(* CoDeSys 2.3 library: TcNciUtilities.lib *)
(* Libraries: TcNci.lib 16.11.12 16:23:10, TcMC.lib 18.1.10 08:53:12, TcBaseMath.lib 27.7.04 11:07:56, TcMath.lib 23.9.04 14:15:30, TcNC.lib 10.10.08 16:55:34, TcIoFunctions.lib 21.7.11 16:19:20, TcUtilities.lib 2.3.12 18:25:40, TcSystem.lib 27.2.12 14:08:36, TcBase.lib 14.5.09 11:14:08, standard.lib 5.6.98 11:03:02, TcNcCfg.lib 22.9.03 17:16:34 *)

(* POU MAIN, ST *)
PROGRAM MAIN
VAR
END_VAR
;
END_PROGRAM

(* POU F_GetVersionTcNciUtilities, ST *)
FUNCTION F_GetVersionTcNciUtilities : UINT
VAR_INPUT
	nVersionElement	: INT;
END_VAR
(*
	Possible nVersionElement parameter:
	1	:	major number
	2	:	minor number
	3	:	revision number
*)
(* Version history:
Date        | Version   | created with							| Author				| Remark
-----------------------------------------------------------------------------------------------------------------------------------------------------------------------------------------------------------------
2013-01-10  | 1.0.3     | TC 2.11								| bw					| Default ADS timeout added
-----------------------------------------------------------------------------------------------------------------------------------------------------------------------------------------------------------------
2013-01-10  | 1.0.2     | TC 2.11 saved as 2.11 Lib		| kbn					| 
-----------------------------------------------------------------------------------------------------------------------------------------------------------------------------------------------------------------
2003-10-07  | 1.0.1     | TC 2.9 B947 saved as 2.8 Lib	| kbn					| lib includes
-----------------------------------------------------------------------------------------------------------------------------------------------------------------------------------------------------------------
2003-09-02  | 1.0.0     | TC 2.9 B947 saved as 2.8 Lib	| Christoph C.		| first release
-----------------------------------------------------------------------------------------------------------------------------------------------------------------------------------------------------------------
*)
CASE nVersionElement OF
1:	(* major number *)
	F_GetVersionTcNciUtilities := 1;
2:	(* minor number *)
	F_GetVersionTcNciUtilities := 0;
3:	(* revision number *)
	F_GetVersionTcNciUtilities := 3;
ELSE
	F_GetVersionTcNciUtilities := 16#FFFF;
END_CASE
END_FUNCTION

(* POU ItpPpgAppendGenericBlock, ST *)
(* Name:       ItpPpgAppendGenericBlock                     *)
(* Desc:       append generic block to the part program     *)
(*             this is just a beta implementation & subject *)
(*             to change                                    *)
(* Author:     kbn                                          *)
(* Date:       05-November-2002                             *)
(* Revision:   VER 1.0.1                                    *)
(* last edit:	VER 1.0.3                                    *)
(*==========================================================*)

FUNCTION_BLOCK ItpPpgAppendGenericBlock
VAR_INPUT
	bExecute:	BOOL;
	sPathName:	STRING;	(* contains path & file name *)
	sBlock:		STRING;
	tTimeOut:	TIME	:= DEFAULT_ADS_TIMEOUT;
END_VAR
VAR_OUTPUT
	bBusy:		BOOL;
	bErr:			BOOL;
	nErrId:		UDINT;
END_VAR
VAR
	nState:				UDINT	:= 0;
	nErrState:			UDINT	:= 0;
	hFile:				UINT;
	fbFileOpen:			FB_FileOpen;
	fbFileClose:		FB_FileClose;
	fbFileAppendLine:	FB_FilePuts;
END_VAR
CASE nState OF
0:
	IF bExecute THEN
		bBusy			:= TRUE;
		bErr			:= FALSE;
		nErrId		:= 0;
		nErrState	:= 0;
		hFile			:= 0;

		(* open existing file *)
		fbFileOpen(
			sNetId		:= '',
			sPathName	:= sPathName,
			nMode			:= FOPEN_MODEAPPEND OR FOPEN_MODETEXT,
			ePath			:= PATH_GENERIC,
			bExecute		:= TRUE,
			tTimeout		:= tTimeOut );

		nState	:= 10;
	END_IF

10:
	(* open existing file *)
	fbFileOpen();

	IF NOT fbFileOpen.bBusy THEN
		fbFileOpen( bExecute := FALSE );
		IF NOT fbFileOpen.bError THEN
			hFile	:= fbFileOpen.hFile;

			(* append line *)
			fbFileAppendLine(
				sNetId	:= '',
				hFile		:= hFile,
				sLine		:= sBlock,
				bExecute	:= TRUE,
				tTimeout	:= tTimeOut );

			nState	:= 20;
		ELSE
			bErr		:= TRUE;
			nErrId	:= fbFileOpen.nErrId;
			nErrState:= nState;
			nState	:= 9999;
		END_IF
	END_IF

20:
	(* append line *)
	fbFileAppendLine();

	IF NOT fbFileAppendLine.bBusy THEN
		fbFileAppendLine( bExecute := FALSE );
		IF NOT fbFileAppendLine.bError THEN
			fbFileClose(
				sNetId	:= '',
				hFile		:= hFile,
				bExecute	:= TRUE,
				tTimeout	:= tTimeOut );
			nState	:= 30;
		ELSE
			bErr		:= TRUE;
			nErrId	:= fbFileAppendLine.nErrId;
			nErrState	:= nState;
			nState	:= 30;	(* we have to close the file anyway *)
		END_IF
	END_IF

30:
	(* close file again *)
	fbFileClose(
		sNetId	:= '',
		hFile		:= hFile,
		bExecute	:= TRUE,
		tTimeout	:= tTimeOut );

	IF NOT fbFileClose.bBusy THEN
		fbFileClose( bExecute := FALSE );
		IF NOT fbFileClose.bError THEN
			IF NOT bExecute THEN
				nState	:= 0;
			ELSE
				nState	:= 9999;
			END_IF
			bBusy	:= FALSE;
		ELSE
			bErr		:= TRUE;
			nErrId	:= fbFileClose.nErrId;
			nErrState:= nState;
			nState	:= 9999;
		END_IF
	END_IF

9999:
	fbFileOpen( bExecute := FALSE );
	fbFileAppendLine( bExecute := FALSE );
	fbFileClose( bExecute := FALSE );

	bBusy	:= FALSE;

	IF NOT bExecute THEN
		nState	:= 0;
	END_IF


END_CASE
END_FUNCTION_BLOCK

(* POU ItpPpgAppendGeoCircleByRadius, ST *)
(* Name:       ItpPpgAppendGeoCircleByRadius                *)
(* Desc:       append a  circle to part program             *)
(*             this is just a beta implementation & subject *)
(*             to change                                    *)
(* Author:     kbn                                          *)
(* Date:       05-November-2002                             *)
(* Revision:   VER 1.0.1                                    *)
(* last edit:	VER 1.0.3                                    *)
(*==========================================================*)

FUNCTION_BLOCK ItpPpgAppendGeoCircleByRadius
VAR_INPUT
	bExecute:		BOOL;
	sPathName:		STRING;	(* contains path & file name *)
	bClockWise:		BOOL;
	fTargetXPos:	LREAL;
	fTargetYPos:	LREAL;
	fTargetZPos:	LREAL;
	fRadius:			LREAL;
	fPathVelo:		LREAL;
	nBlockNo:		UDINT;
	tTimeOut:		TIME	:= DEFAULT_ADS_TIMEOUT;
END_VAR
VAR_OUTPUT
	bBusy:		BOOL;
	bErr:			BOOL;
	nErrId:		UDINT;
END_VAR
VAR
	nState:				UDINT	:= 0;
	fbFormatString:	FB_FormatString;
	sBlock:				T_MaxString;
	fbAppendBlock:		ItpPpgAppendGenericBlock;
	fBlockNo:			LREAL;
END_VAR
CASE nState OF

0:
	IF bExecute THEN
		bBusy		:= TRUE;
		bErr		:= FALSE;
		nErrId	:= 0;

		fBlockNo	:= UDINT_TO_LREAL( nBlockNo );

		IF bClockWise THEN
			fbFormatString(
				sFormat:= 'N%.0f G2 X%.3f Y%.3f Z%.3f B%.3f F%.3f $N',
				arg1:= F_LREAL( fBlockNo ),
				arg2:= F_LREAL( fTargetXPos ),
				arg3:= F_LREAL( fTargetYPos ),
				arg4:= F_LREAL( fTargetZPos ),
				arg5:= F_LREAL( fRadius ),
				arg6:= F_LREAL( fPathVelo ) );
		ELSE
			fbFormatString(
				sFormat:= 'N%.0f G3 X%.3f Y%.3f Z%.3f B%.3f F%.3f $N',
				arg1:= F_LREAL( fBlockNo ),
				arg2:= F_LREAL( fTargetXPos ),
				arg3:= F_LREAL( fTargetYPos ),
				arg4:= F_LREAL( fTargetZPos ),
				arg5:= F_LREAL( fRadius ),
				arg6:= F_LREAL( fPathVelo ) );
		END_IF

		IF NOT fbFormatString.bError THEN
			sBlock	:= fbFormatString.sOut;

			nState	:= 10;
		ELSE
			bErr		:= TRUE;
			nErrId	:= fbFormatString.nErrId;

			nState	:= 9999;
		END_IF

	END_IF

10:
	fbAppendBlock(
		bExecute		:= TRUE,
		sPathName	:= sPathName,
		sBlock		:= sBlock,
		tTimeOut		:= tTimeOut );

	IF NOT fbAppendBlock.bBusy THEN
		fbAppendBlock( bExecute := FALSE );

		IF NOT fbAppendBlock.bErr THEN
			bBusy	:= FALSE;
			IF NOT bExecute THEN
				nState	:= 0;
			ELSE
				nState	:= 9999;
			END_IF
		ELSE
			(* an error occured *)
			bErr		:= TRUE;
			nErrId	:= fbAppendBlock.nErrId;
			nState	:= 9999;
		END_IF

	END_IF

9999:
	bBusy	:= FALSE;
	fbAppendBlock( bExecute := FALSE );

	IF NOT bExecute THEN
		nState	:= 0;
	END_IF

END_CASE
END_FUNCTION_BLOCK

(* POU ItpPpgAppendGeoLine, ST *)
(* Name:       ItpPpgAppendGeoLine                          *)
(* Desc:       append a line to the part program            *)
(*             this is just a beta implementation & subject *)
(*             to change                                    *)
(* Author:     kbn                                          *)
(* Date:       05-November-2002                             *)
(* Revision:   VER 1.0.1                                    *)
(* last edit:	VER 1.0.3                                    *)
(*==========================================================*)

FUNCTION_BLOCK ItpPpgAppendGeoLine
VAR_INPUT
	bExecute:		BOOL;
	sPathName:		STRING;	(* contains path & file name *)
	fTargetXPos:	LREAL;
	fTargetYPos:	LREAL;
	fTargetZPos:	LREAL;
	fPathVelo:		LREAL;
	nBlockNo:		UDINT;
	tTimeOut:		TIME	:= DEFAULT_ADS_TIMEOUT;
END_VAR
VAR_OUTPUT
	bBusy:		BOOL;
	bErr:			BOOL;
	nErrId:		UDINT;
END_VAR
VAR
	nState:				UDINT	:= 0;
	fbFormatString:	FB_FormatString;
	sBlock:				T_MaxString;
	fbAppendToFile:	ItpPpgAppendGenericBlock;
	fBlockNo:			LREAL;
	hFile:				UINT;
END_VAR
CASE nState OF

0:
	IF bExecute THEN
		bBusy		:= TRUE;
		bErr		:= FALSE;
		nErrId	:= 0;

		fBlockNo	:= UDINT_TO_LREAL( nBlockNo );

		fbFormatString(
			sFormat:= 'N%.0f G1 X%.3f Y%.3f Z%.3f F%.3f $N',
			arg1:= F_LREAL( fBlockNo ),
			arg2:= F_LREAL( fTargetXPos ),
			arg3:= F_LREAL( fTargetYPos ),
			arg4:= F_LREAL( fTargetZPos ),
			arg5:= F_LREAL( fPathVelo ) );

		IF NOT fbFormatString.bError THEN
			sBlock	:= fbFormatString.sOut;

			nState	:= 10;
		ELSE
			bErr		:= TRUE;
			nErrId	:= fbFormatString.nErrId;

			nState	:= 9999;
		END_IF

	END_IF

10:
	fbAppendToFile(
		bExecute		:= TRUE,
		sPathName	:= sPathName,
		sBlock		:= sBlock,
		tTimeOut		:= tTimeOut );

	IF NOT fbAppendToFile.bBusy THEN
		fbAppendToFile( bExecute := FALSE );

		IF NOT fbAppendToFile.bErr THEN
			IF NOT bExecute THEN
				nState	:= 0;
			ELSE
				nState	:= 9999;
			END_IF
			bBusy	:= FALSE;
		ELSE
			bErr		:= TRUE;
			nErrId	:= fbAppendToFile.nErrId;
			nState	:= 9999;
		END_IF
	END_IF

9999:
	bBusy	:= FALSE;
	fbAppendToFile( bExecute := FALSE );

	IF NOT bExecute THEN
		nState	:= 0;
	END_IF

END_CASE
END_FUNCTION_BLOCK

(* POU ItpPpgCloseMain, ST *)
(* Name:       ItpPpgCloseMain                              *)
(* Desc:       generate code for part program end (M02)     *)
(*             this is just a beta implementation & subject *)
(*             to change                                    *)
(* Author:     kbn                                          *)
(* Date:       05-November-2002                             *)
(* Revision:   VER 1.0.1                                    *)
(* last edit:	VER 1.0.3                                    *)
(*==========================================================*)

FUNCTION_BLOCK ItpPpgCloseMain
VAR_INPUT
	bExecute:	BOOL;
	sPathName:	STRING;	(* contains path & file name *)
	tTimeOut:	TIME	:= DEFAULT_ADS_TIMEOUT;
END_VAR
VAR_OUTPUT
	bBusy:		BOOL;
	bErr:			BOOL;
	nErrId:		UDINT;
END_VAR
VAR
	fbAppendBlock:	ItpPpgAppendGenericBlock;
END_VAR
fbAppendBlock(
	bExecute		:= bExecute,
	sPathName	:= sPathName,
	sBlock		:= 'M02$N',
	tTimeOut		:= tTimeOut );

bBusy		:= fbAppendBlock.bBusy;
bErr		:= fbAppendBlock.bErr;
nErrId	:= fbAppendBlock.nErrId;
END_FUNCTION_BLOCK

(* POU ItpPpgCloseSubroutine, ST *)
(* Name:       ItpPpgCloseSubroutine                        *)
(* Desc:       generate code for subroutine end (M17)       *)
(*             this is just a beta implementation & subject *)
(*             to change                                    *)
(* Author:     kbn                                          *)
(* Date:       05-November-2002                             *)
(* Revision:   VER 1.0.1                                    *)
(* last edit:	VER 1.0.3                                    *)
(*==========================================================*)

FUNCTION_BLOCK ItpPpgCloseSubroutine
VAR_INPUT
	bExecute:	BOOL;
	sPathName:	STRING;	(* contains path & file name *)
	tTimeOut:	TIME	:= DEFAULT_ADS_TIMEOUT;
END_VAR
VAR_OUTPUT
	bBusy:		BOOL;
	bErr:			BOOL;
	nErrId:		UDINT;
END_VAR
VAR
	fbAppendBlock:	ItpPpgAppendGenericBlock;
END_VAR
(* generate M17 *)

fbAppendBlock(
	bExecute		:= bExecute,
	sPathName	:= sPathName,
	sBlock		:= 'M17$N',
	tTimeOut		:= tTimeOut );

bBusy		:= fbAppendBlock.bBusy;
bErr		:= fbAppendBlock.bErr;
nErrId	:= fbAppendBlock.nErrId;
END_FUNCTION_BLOCK

(* POU ItpPpgCreateMain, ST *)
(* Name:       ItpPpgCreateMain                             *)
(* Desc:       creates empty file for the part program      *)
(*             this is just a beta implementation & subject *)
(*             to change                                    *)
(* Author:     kbn                                          *)
(* Date:       05-November-2002                             *)
(* Revision:   VER 1.0.1                                    *)
(* last edit:	VER 1.0.3                                    *)
(*==========================================================*)

FUNCTION_BLOCK ItpPpgCreateMain
VAR_INPUT
	bExecute:	BOOL;
	sPathName:	STRING;	(* contains path & file name *)
	tTimeOut:	TIME	:= DEFAULT_ADS_TIMEOUT;
END_VAR
VAR_OUTPUT
	bBusy:		BOOL;
	bErr:			BOOL;
	nErrId:		UDINT;
END_VAR
VAR
	nState:		UDINT	:= 0;
	nErrState:	UDINT	:= 0;
	hFile:			UINT;
	fbFileOpen:		FB_FileOpen;
	fbFileClose:	FB_FileClose;
	fbFileAppendLine:	FB_FilePuts;
END_VAR
CASE nState OF
0:
	IF bExecute THEN
		bBusy		:= TRUE;
		bErr		:= FALSE;
		nErrId	:= 0;
		nErrState	:= 0;
		hFile			:= 0;

		nState	:= 10;
	END_IF

10:
	(* create & open file *)
	fbFileOpen(
		sNetId		:= '',
		sPathName	:= sPathName,
		nMode			:= FOPEN_MODEWRITE OR FOPEN_MODETEXT ,
		ePath			:= PATH_GENERIC,
		bExecute		:= TRUE,
		tTimeout		:= tTimeOut );

	IF NOT fbFileOpen.bBusy THEN
		fbFileOpen( bExecute := FALSE );
		IF NOT fbFileOpen.bError THEN
			hFile	:= fbFileOpen.hFile;
			nState	:= 20;
		ELSE
			bErr		:= TRUE;
			nErrId	:= fbFileOpen.nErrId;
			nErrState:= nState;
			nState	:= 9999;
		END_IF
	END_IF

20:
	(* write header *)
	fbFileAppendLine(
		sNetId	:= '',
		hFile		:= hFile,
		sLine		:= '(this file is created by ppg)$N',
		bExecute	:= TRUE,
		tTimeout	:= tTimeOut );

	IF NOT fbFileAppendLine.bBusy THEN
		fbFileAppendLine( bExecute := FALSE );
		IF NOT fbFileAppendLine.bError THEN
			nState	:= 30;
		ELSE
			bErr			:= TRUE;
			nErrId		:= fbFileAppendLine.nErrId;
			nErrState	:= nState;
			(* we still have to close the file - so goto state 30 *)
			nState	:= 30;
		END_IF
	END_IF

30:

	fbFileClose(
		sNetId	:= '',
		hFile		:= hFile,
		bExecute	:= TRUE,
		tTimeout	:= tTimeOut );

	IF NOT fbFileClose.bBusy THEN
		fbFileClose( bExecute := FALSE );
		IF NOT fbFileClose.bError THEN
			IF NOT bExecute THEN
				nState	:= 0;
			ELSE
				nState	:= 9999;
			END_IF
			bBusy	:= FALSE;
		ELSE
			bErr		:= TRUE;
			nErrId	:= fbFileClose.nErrId;
			nErrState:= nState;
			nState	:= 9999;
		END_IF
	END_IF

9999:
	bBusy	:= FALSE;

	fbFileClose( bExecute := FALSE );
	fbFileOpen( bExecute := FALSE );
	fbFileAppendLine( bExecute := FALSE );

	IF NOT bExecute THEN
		nState	:= 0;
	END_IF
END_CASE
END_FUNCTION_BLOCK

(* POU ItpPpgCreateSubroutine, ST *)
(* Name:       ItpPpgCreateSubroutine                       *)
(* Desc:       creates empty file for the subroutine        *)
(*             this is just a beta implementation & subject *)
(*             to change                                    *)
(* Author:     kbn                                          *)
(* Date:       05-November-2002                             *)
(* Revision:   VER 1.0.1                                    *)
(* last edit:	VER 1.0.3                                    *)
(*==========================================================*)

FUNCTION_BLOCK ItpPpgCreateSubroutine
VAR_INPUT
	bExecute:			BOOL;
	sPathName:			STRING;	(* contains path & file name with suffix *)
	nSubroutineId:		UDINT;
	tTimeOut:	TIME	:= DEFAULT_ADS_TIMEOUT;
END_VAR
VAR_OUTPUT
	bBusy:		BOOL;
	bErr:			BOOL;
	nErrId:		UDINT;
END_VAR
VAR
	hFile:				UINT;
	nState:				UDINT	:= 0;
	nErrState:			UDINT	:= 0;
	sBlock:				T_MaxString;
	fbFileOpen:			FB_FileOpen;
	fbFileClose:		FB_FileClose;
	fbFileAppendLine:	FB_FilePuts;
	fbFormatString:	FB_FormatString;
	fSubRoutineId:		LREAL;
END_VAR
CASE nState OF
0:
	IF bExecute THEN
		bBusy		:= TRUE;
		bErr		:= FALSE;
		nErrId	:= 0;
		nErrState	:= 0;
		hFile			:= 0;

		nState	:= 10;
	END_IF

10:
	(* create & open file *)
	fbFileOpen(
		sNetId		:= '',
		sPathName	:= sPathName,
		nMode			:= FOPEN_MODEWRITE OR FOPEN_MODETEXT ,
		ePath			:= PATH_GENERIC,
		bExecute		:= TRUE,
		tTimeout		:= tTimeOut );

	IF NOT fbFileOpen.bBusy THEN
		IF NOT fbFileOpen.bError THEN
			hFile	:= fbFileOpen.hFile;
			fbFileOpen( bExecute := FALSE );
			nState	:= 20;
		ELSE
			bErr		:= TRUE;
			nErrId	:= fbFileOpen.nErrId;
			nErrState:= nState;
			nState	:= 9999;
		END_IF
	END_IF

20:
	(* write header *)
	fbFileAppendLine(
		sNetId	:= '',
		hFile		:= hFile,
		sLine		:= '(this file is created by ppg)$N',
		bExecute	:= TRUE,
		tTimeout	:= tTimeOut );

	IF NOT fbFileAppendLine.bBusy THEN
		fbFileAppendLine( bExecute := FALSE );
		IF NOT fbFileAppendLine.bError THEN
			nState	:= 30;
		ELSE
			bErr			:= TRUE;
			nErrId		:= fbFileAppendLine.nErrId;
			nErrState	:= nState;
			(* we still have to close the file - so goto state 1000 *)
			nState	:= 1000;
		END_IF
	END_IF

30:
		fSubRoutineId	:= UDINT_TO_REAL( nSubroutineId );

		fbFormatString(
			sFormat:= 'L%.0f$N',
			arg1:= F_LREAL( fSubRoutineId ) );

		IF NOT fbFormatString.bError THEN
			sBlock	:= fbFormatString.sOut;
			nState	:= 40;
		ELSE
			bErr		:= TRUE;
			nErrId	:= fbFormatString.nErrId;
			(* we still have to close the file - so goto state 1000 *)
			nState	:= 1000;
		END_IF

40:
	fbFileAppendLine(
		sNetId	:= '',
		hFile		:= hFile,
		sLine		:= sBlock,
		bExecute	:= TRUE,
		tTimeout	:= tTimeOut );

	IF NOT fbFileAppendLine.bBusy THEN
		fbFileAppendLine( bExecute := FALSE );
		IF NOT fbFileAppendLine.bError THEN
			nState	:= 1000;
		ELSE
			bErr			:= TRUE;
			nErrId		:= fbFileAppendLine.nErrId;
			nErrState	:= nState;
			(* we still have to close the file - so goto state 1000 *)
			nState	:= 1000;
		END_IF
	END_IF

1000:
	(* close file *)
	IF hFile <> 0 THEN
		fbFileClose(
			sNetId	:= '',
			hFile		:= hFile,
			bExecute	:= TRUE,
			tTimeout	:= tTimeOut );
	END_IF
	nState	:= 1010;

1010:
	fbFileClose();

	IF NOT fbFileClose.bBusy THEN
		fbFileClose( bExecute := FALSE );
		IF NOT fbFileClose.bError THEN
			IF NOT bExecute THEN
				nState	:= 0;
			ELSE
				nState	:= 9999;
			END_IF
			bBusy	:= FALSE;
		ELSE
			bErr		:= TRUE;
			nErrId	:= fbFileClose.nErrId;
			nErrState:= nState;
			nState	:= 9999;
		END_IF
	END_IF

9999:
	bBusy	:= FALSE;

	fbFileClose( bExecute := FALSE );
	fbFileOpen( bExecute := FALSE );
	fbFileAppendLine( bExecute := FALSE );

	IF NOT bExecute THEN
		nState	:= 0;
	END_IF
END_CASE
END_FUNCTION_BLOCK
